// TwinCAT 3 PLC project PlcConveyor
// ProgramVersion: 3.1.4024.0
// project tree:
//   POUs/ MAIN.TcPOU

// ---- POUs/MAIN.TcPOU
PROGRAM MAIN
VAR
    running : BOOL;
    statusText : STRING;
END_VAR

running := TRUE;
statusText := BOOL_TO_STRING(running);

END_PROGRAM
